FUNCTION TFConsentiDepositoPaccoSuWA : BOOL // Valuta se esiste una WA in lavorazione con lo stesso codice, se esiste ritorna false, altrimenti true
VAR_INPUT
	WorkArea : POINTER TO ARRAY [1..MAXAREA] OF TFMachinePalletizer_WorkArea;
	WorkAreaState : POINTER TO ARRAY [1..MAXAREA] OF TFMachinePalletizer_WorkAreaState;
	NWaInValutazione : INT;
END_VAR
VAR
	wa : INT;
END_VAR

// Valuta se esiste una WA in lavorazione con lo stesso codice, se esiste ritorna false, altrimenti true
TFConsentiDepositoPaccoSuWA := TRUE;

(* Per tutte le WorkArea Attive e in Lavorazione *)
FOR wa:=1 TO MAXAREAPRESENT DO
	IF wa <> NWaInValutazione THEN
		IF WorkArea^[wa].Enable = 1 THEN
		(* Verifico se è in lavorazione *)
			IF WorkAreaState^[wa].State = WORKAREA_STATE_OCCUPIED_WORKING THEN
				(* Verifico se il codice è uguale *)
				IF WorkAreaState^[wa].Code = WorkAreaState^[NWaInValutazione].Code THEN
					(* Verifico se ha già dei pacchi depositati *)
					IF WorkAreaState^[wa].P > WorkAreaState^[NWaInValutazione].P AND WorkAreaState^[NWaInValutazione].P <>-1  THEN 
						TFConsentiDepositoPaccoSuWA := FALSE;
						RETURN;
					END_IF
				END_IF
			END_IF
		END_IF
	END_IF
END_FOR

END_FUNCTION

(* stored: Version 1.1.0.1, ProductVersion 3.1.4024.11
   POU TFConsentiDepositoPaccoSuWA: Id {aaaccde4-a6a9-46e9-ad33-9c666e586899}, SpecialFunc None *)
